PROGRAM AzimuthControl
VAR_INPUT
	left:	BOOL;
	right: BOOL;
	reset: BOOL;
	enable :  BOOL;
END_VAR

VAR
	AzimuthAxisJog:	FB_AxisJog;
	AzimuthAxis:		FB_Axis2;
	error: BOOL;
	ErrorID: UDINT;
	position: LREAL;
	act_position: LREAL;
	AzimuthAxisEvent: FB_EventLog;
END_VAR

IF PendantControl.manual THEN
	AzimuthAxisJog(	bPowerEnable := enable AND Main.power_OK,
						bEnable_Positive := GVL_Telescope.brake_azimuth_eve,
						bEnable_Negative := GVL_Telescope.brake_azimuth_eve,
						bForward := left,
						bBackward := right,
						bReset := reset,
						bStop := left AND right,
						bErr => error,
						fActPos => act_position,
						stAxis :=	GVL_Telescope.AzimuthAxisRef);	
ELSE
	AzimuthAxis(	Enable := TelescopeControl.power AND Main.power_OK,
					Reset := reset,
					Position := position, 
					ActualPosition => act_position,
					Error => error,
					ErrorID => ErrorID,
					AxisRef :=	GVL_Telescope.AzimuthAxisRef);
END_IF

AzimuthAxisEvent(	Trigger := Error, 
				Level := ADSLOG_MSGTYPE_ERROR,
				FormatString := 'Azimuth Axis Error: %s',
				OnMessage := UDINT_TO_STRING(ErrorID),
				OffMEssage := 'OK');

END_PROGRAM

(* stored: Version 1.1.0.1, ProductVersion 3.1.4024.4
   POU AzimuthControl: Id {8e08648a-b748-4448-9dcc-aa13dfcf6a06}, SpecialFunc None *)
